# B&R Automation Studio project LAB_1
Automation Studio 4.5.2.102

## Configuration Config1

### Hardware
```
4PP065_0351_P74 : 4PP065.0351-P74 v1.0.4.0
  Connector IF5:
    ActivateDevice = 1
  ConfigurationID = LAB_1_1_Config1
  Simulation = 1
  KeyMappingFile = VC\4PP065_0351_P74.dis
```

## Logical view

Binary libraries used (declarations not repeated): Library

### Program Logical/Program

#### Variables.var
```iecst
VAR
	fb_regulator : {REDUND_UNREPLICABLE} FB_Regulator;
	fb_motor_1 : {REDUND_UNREPLICABLE} FB_Motor;
	fb_motor_2 : {REDUND_UNREPLICABLE} FB_Motor;
	speed : {REDUND_UNREPLICABLE} REAL;
	enable : {REDUND_UNREPLICABLE} BOOL;
	counter : {REDUND_UNREPLICABLE} REAL;
END_VAR
```

#### Main.c
```c
#include <bur/plctypes.h>

#ifdef _DEFAULT_INCLUDES
	#include <AsDefault.h>
#endif

void _INIT ProgramInit(void)
{
	enable = 1;
	counter = 0;
	speed = 0;
	fb_regulator.dt = 0.02;
	fb_regulator.k_i = 16;
	fb_regulator.k_p = 0.64;
	fb_regulator.max_abs_value = 24;
	fb_motor_1.dt = 0.02;
	fb_motor_1.ke = 16;
	fb_motor_1.Tm = 0.04;
	fb_motor_2.dt = 0.02;
	fb_motor_2.ke = 16;
	fb_motor_2.Tm = 0.04;

}

void _CYCLIC ProgramCyclic(void)
{
	if(enable == 1)
	{
		counter += 10;
		if(counter >= 1000 && counter <= 1500) speed = 5;
		else speed = 0;
	}
	else speed = 0;
	fb_regulator.e = speed - fb_motor_1.w;
	FB_Regulator(&(fb_regulator));
	fb_motor_1.u = fb_regulator.u*fb_motor_1.ke;
	fb_motor_2.u = speed*fb_motor_2.ke;
	FB_Motor(&(fb_motor_1));
	FB_Motor(&(fb_motor_2));

}

void _EXIT ProgramExit(void)
{

}
```
